// TwinCAT 3 PLC project Machine
// Title: test
// Company: test
// ProjectVersion: 1.1
// ProgramVersion: 3.1.4022.1
// libraries:
//   GWP Library, * (Viessmann)
//   Tc2_Standard, * (Beckhoff Automation GmbH)
//   Tc2_System, * (Beckhoff Automation GmbH)
//   Tc3_Module, * (Beckhoff Automation GmbH)
//   VisuDialogs, * (System)
//   VisuSymbols, * (System)
//   VisuSymbols,3.5.10.0,System
// project tree:
//   / GlobalTextList.TcGTLO, PlcTask.TcTTO, VisualizationManager.TcVMO (not stored), VISU_TASK.TcTTO
//   POUs/ IOs.TcPOU, Main.TcPOU
//   VISUs/ Infoseite.TcVIS, Alarmliste.TcVIS, Fusszeile_50.TcVIS, Test_Login.TcVIS, Testkachel.TcVIS
//   VISUs/Benutzerebene/ Login.TcVIS
//   VISUs/Betriebsarten/Wärmegewinnung/KWP/ KWP_SP_AC_NC_CLK_D.TcVIS, KWP_SP_AC_NC.TcVIS, KWP_SP_AC_NC_GR_4_ohne_RE.TcVIS, KWP_SP_AC_NC_Sollwerte.TcVIS, KWP_SP_AC_NC_PU_Sollwerte.TcVIS
//   VISUs/Betriebsarten/Wärmegewinnung/VD/ VD_Sollwerte_zuruecksetzen.TcVIS, VD.TcVIS, VD_GW_Sollwerte.TcVIS, VD_PU_Sollwerte.TcVIS, VD_VTL_Sollwerte.TcVIS
//   VISUs/Betriebsarten/Wärmesenke/HWP_SP/ HWP_SP.TcVIS, HWP_SP_CLK_D.TcVIS, HWP_SP_GR_4_ohne_RE.TcVIS, HWP_SP_Sollwerte.TcVIS
//   VISUs/Betriebsarten/Wärmesenke/KD/ KD.TcVIS, KD_PU_Sollwerte.TcVIS, KD_Sollwerte_zuruecksetzen.TcVIS, KD_VTL_Sollwerte.TcVIS
//   VISUs/Betriebsarten/Wärmesenke/TWW_SP/ TWW_SP.TcVIS, TWW_SP_CLK_I_Zwangsladung_1.TcVIS, TWW_SP_Sollwerte.TcVIS, TWW_SP_CLK_I_Zwangsladung_2.TcVIS, TWW_SP_PU_Sollwerte.TcVIS
//   VISUs/Betriebsarten/Wärmesenke/Zirkulationspumpe/ Zirkulationspumpe_Sollwerte.TcVIS, Zirkulationspumpe_CLK_W7_Siebentageprogramm.TcVIS
//   VISUs/Betriebsarten/Wärmesenke/Zusatzheizung/ Zusatzheizung_Sollwerte.TcVIS
//   VISUs/Hauptmenu/ Hauptmenu.TcVIS
//   VISUs/Home/ Home.TcVIS
//   VISUs/Maschine/ EG_Innen.TcVIS, EEv.TcVIS, Kreis_3KO_SollwerteAllg.TcVIS, Kreis_3KO.TcVIS
//   VISUs/Sollwertmenu/ Sollwertmenu.TcVIS, Sollwertmenu_Zirk_PU.TcVIS, Sollwertmenu_Waermegewinnung.TcVIS, Sollwertmenu_Waermepumpe.TcVIS, Sollwertmenu_KWP.TcVIS, Sollwertmenu_Waermesenke.TcVIS, Sollwertmenu_KD.TcVIS, Sollwertmenu_HWP.TcVIS, Sollwertmenu_TWW.TcVIS
// real-time tasks:
//   TASK PlcTask: cycle T#10ms, priority 20, ADS port 350
//   TASK VISU_TASK: cycle T#200000us, priority 30, ADS port 351
// I/O:
//   DEVICE Device 1 (EtherCAT), AmsNetId 5.52.29.192.2.1
//     Term 1 (EK1100) [EK1100 EtherCAT Coupler (2A E-Bus)]
//       Term 2 (EL1809) [EL1809 16Ch. Dig. Input 24V, 3ms]
//       Term 3 (EL2809) [EL2809 16Ch. Dig. Output 24V, 0.5A]
//       Term 4 (EL3208) [EL3208 8Ch. Ana. Input PT100 (RTD)]
//       Term 5 (EL3208) [EL3208 8Ch. Ana. Input PT100 (RTD)]
//       Term 6 (EL3058) [EL3058 8Ch. Ana. Input 4-20mA]
//       Term 7 (EL4008) [EL4008 8Ch. Ana. Output 0-10V, 12bit]
//       Term 8 (EL7031) [EL7031 1Ch. Stepper motor output stage (24V, 1.5A)]
//       Term 9 (EL1809) [EL1809 16Ch. Dig. Input 24V, 3ms]
//       Term 10 (EL1809) [EL1809 16Ch. Dig. Input 24V, 3ms]
//       Term 11 (EL2809) [EL2809 16Ch. Dig. Output 24V, 0.5A]
//       Term 12 (EL2809) [EL2809 16Ch. Dig. Output 24V, 0.5A]
//       Term 13 (EL3208) [EL3208 8Ch. Ana. Input PT100 (RTD)]
//       Term 14 (EL3208) [EL3208 8Ch. Ana. Input PT100 (RTD)]
//       Term 15 (EL4008) [EL4008 8Ch. Ana. Output 0-10V, 12bit]
//       Term 16 (EL3208) [EL3208 8Ch. Ana. Input PT100 (RTD)]
//       Term 17 (EL3403-0010) [EL3403-0010 3Ch. Power Measuring, 5A]
//       Term 18 (EL9011) [EL9011 End Terminal]
// variable links:
//   Machine/Machine Instance <-> Device 1 (EtherCAT)/Term 1 (EK1100)/Term 10 (EL1809)
//     PlcTask Inputs/Main.IOs_0.DI_851KF1.ix_DI{1..16} <-> Channel {1..16}/Input  (16 links)
//   Machine/Machine Instance <-> Device 1 (EtherCAT)/Term 1 (EK1100)/Term 11 (EL2809)
//     PlcTask Outputs/Main.IOs_0.DO_851KF2.qx_DO{1..16} <-> Channel {1..16}/Output  (16 links)
//   Machine/Machine Instance <-> Device 1 (EtherCAT)/Term 1 (EK1100)/Term 12 (EL2809)
//     PlcTask Outputs/Main.IOs_0.DO_851KF2_1.qx_DO{1..16} <-> Channel {1..16}/Output  (16 links)
//   Machine/Machine Instance <-> Device 1 (EtherCAT)/Term 1 (EK1100)/Term 13 (EL3208)
//     PlcTask Inputs/Main.IOs_0.AI_851KF3.ii_AI{1..8} <-> RTD Inputs Channel {1..8}/Value  (8 links)
//   Machine/Machine Instance <-> Device 1 (EtherCAT)/Term 1 (EK1100)/Term 14 (EL3208)
//     PlcTask Inputs/Main.IOs_0.AI_851KF4.ii_AI{1..8} <-> RTD Inputs Channel {1..8}/Value  (8 links)
//   Machine/Machine Instance <-> Device 1 (EtherCAT)/Term 1 (EK1100)/Term 15 (EL4008)
//     PlcTask Outputs/Main.IOs_0.AO_851KF4_1.qi_AO{1..8} <-> AO Outputs Channel {1..8}/Analog output  (8 links)
//   Machine/Machine Instance <-> Device 1 (EtherCAT)/Term 1 (EK1100)/Term 16 (EL3208)
//     PlcTask Inputs/Main.IOs_0.AI_851KF6.ii_AI{1..8} <-> RTD Inputs Channel {1..8}/Value  (8 links)
//   Machine/Machine Instance <-> Device 1 (EtherCAT)/Term 1 (EK1100)/Term 17 (EL3403-0010)
//     PlcTask Inputs/Main.IOs_0.EM_851KF6_1.ii_ActivePower_L1 <-> PM Inputs Channel 1/Active power
//     PlcTask Inputs/Main.IOs_0.EM_851KF6_1.ii_ActivePower_L2 <-> PM Inputs Channel 2/Active power
//     PlcTask Inputs/Main.IOs_0.EM_851KF6_1.ii_ActivePower_L3 <-> PM Inputs Channel 3/Active power
//     PlcTask Inputs/Main.IOs_0.EM_851KF6_1.ii_Current_L1 <-> PM Inputs Channel 1/Current
//     PlcTask Inputs/Main.IOs_0.EM_851KF6_1.ii_Current_L2 <-> PM Inputs Channel 2/Current
//     PlcTask Inputs/Main.IOs_0.EM_851KF6_1.ii_Current_L3 <-> PM Inputs Channel 3/Current
//     PlcTask Inputs/Main.IOs_0.EM_851KF6_1.ii_Index_L1 <-> PM Inputs Channel 1/Index
//     PlcTask Inputs/Main.IOs_0.EM_851KF6_1.ii_Index_L2 <-> PM Inputs Channel 2/Index
//     PlcTask Inputs/Main.IOs_0.EM_851KF6_1.ii_Index_L3 <-> PM Inputs Channel 3/Index
//     PlcTask Inputs/Main.IOs_0.EM_851KF6_1.ii_VariantValue_L1 <-> PM Inputs Channel 1/Variant value
//     PlcTask Inputs/Main.IOs_0.EM_851KF6_1.ii_VariantValue_L2 <-> PM Inputs Channel 2/Variant value
//     PlcTask Inputs/Main.IOs_0.EM_851KF6_1.ii_VariantValue_L3 <-> PM Inputs Channel 3/Variant value
//     PlcTask Inputs/Main.IOs_0.EM_851KF6_1.ii_Voltage_L1 <-> PM Inputs Channel 1/Voltage
//     PlcTask Inputs/Main.IOs_0.EM_851KF6_1.ii_Voltage_L2 <-> PM Inputs Channel 2/Voltage
//     PlcTask Inputs/Main.IOs_0.EM_851KF6_1.ii_Voltage_L3 <-> PM Inputs Channel 3/Voltage
//     PlcTask Outputs/Main.IOs_0.EM_851KF6_1.qi_Index_L1 <-> PM Outputs Channel 1/Index
//     PlcTask Outputs/Main.IOs_0.EM_851KF6_1.qi_Index_L2 <-> PM Outputs Channel 2/Index
//     PlcTask Outputs/Main.IOs_0.EM_851KF6_1.qi_Index_L3 <-> PM Outputs Channel 3/Index
//   Machine/Machine Instance <-> Device 1 (EtherCAT)/Term 1 (EK1100)/Term 2 (EL1809)
//     PlcTask Inputs/Main.IOs_0.DI_850KF2.ix_DI{1..16} <-> Channel {1..16}/Input  (16 links)
//   Machine/Machine Instance <-> Device 1 (EtherCAT)/Term 1 (EK1100)/Term 3 (EL2809)
//     PlcTask Outputs/Main.IOs_0.DO_850KF3.qx_DO{1..16} <-> Channel {1..16}/Output  (16 links)
//   Machine/Machine Instance <-> Device 1 (EtherCAT)/Term 1 (EK1100)/Term 4 (EL3208)
//     PlcTask Inputs/Main.IOs_0.AI_850KF4.ii_AI{1..8} <-> RTD Inputs Channel {1..8}/Value  (8 links)
//   Machine/Machine Instance <-> Device 1 (EtherCAT)/Term 1 (EK1100)/Term 5 (EL3208)
//     PlcTask Inputs/Main.IOs_0.AI_850KF4_1.ii_AI{1..8} <-> RTD Inputs Channel {1..8}/Value  (8 links)
//   Machine/Machine Instance <-> Device 1 (EtherCAT)/Term 1 (EK1100)/Term 6 (EL3058)
//     PlcTask Inputs/Main.IOs_0.AI_850KF5.ii_AI{1..8} <-> AI Standard Channel {1..8}/Value  (8 links)
//   Machine/Machine Instance <-> Device 1 (EtherCAT)/Term 1 (EK1100)/Term 7 (EL4008)
//     PlcTask Outputs/Main.IOs_0.AO_850KF6.qi_AO{1..8} <-> AO Outputs Channel {1..8}/Analog output  (8 links)
//   Machine/Machine Instance <-> Device 1 (EtherCAT)/Term 1 (EK1100)/Term 8 (EL7031)
//     PlcTask Inputs/Main.IOs_0.SM_850KF6_1.ii_CounterValue <-> ENC Status/Counter value
//     PlcTask Outputs/Main.IOs_0.SM_850KF6_1.qi_SetCounter <-> ENC Control/Set counter value
//     PlcTask Outputs/Main.IOs_0.SM_850KF6_1.qi_Velo <-> STM Velocity/Velocity
//     PlcTask Outputs/Main.IOs_0.SM_850KF6_1.qx_EN <-> STM Control/Control/Enable
//     PlcTask Outputs/Main.IOs_0.SM_850KF6_1.qx_SetCounter <-> ENC Control/Control/Set counter
//   Machine/Machine Instance <-> Device 1 (EtherCAT)/Term 1 (EK1100)/Term 9 (EL1809)
//     PlcTask Inputs/Main.IOs_0.DI_851KF0.ix_DI{1..16} <-> Channel {1..16}/Input  (16 links)

CONFIGURATION Machine
    RESOURCE PLC ON TwinCAT3
        TASK PlcTask(INTERVAL := T#10ms, PRIORITY := 20);
        TASK VISU_TASK(INTERVAL := T#200000us, PRIORITY := 30);
        PROGRAM Main WITH PlcTask : Main;
        PROGRAM VisuElems_Visu_Prg WITH VISU_TASK : VisuElems.Visu_Prg;
    END_RESOURCE
END_CONFIGURATION

// ---- POUs/Main.TcPOU
PROGRAM Main
VAR
	KWP_SP_AC_NC_0: KWP_SP_AC_NC;
	VD_0: VD;
	KD_0: KD;
	Kreis_3KO_0: Kreis_3KO;
	HWP_SP_0: HWP_SP;
	Zusatzheizung_0: Zusatzheizung;
	Zirk_Pumpe_0: Zirk_Pumpe;
	TWW_SP_0: TWW_SP;
	Init_0: Init;
	IOs_0: IOs;
	AI_to_Druck_0: AI_to_Druck;
	AI_to_Druck_1: AI_to_Druck;
	Logger_0: logger;
	Alarme_1bis10: alarm;
	Alarme_11bis20: alarm;
	Alarme_21bis30: alarm;
	Alarmliste_FB_0: Alarmliste_FB;
END_VAR
VAR PERSISTENT
	dut_Liste:SW_Struct;
END_VAR

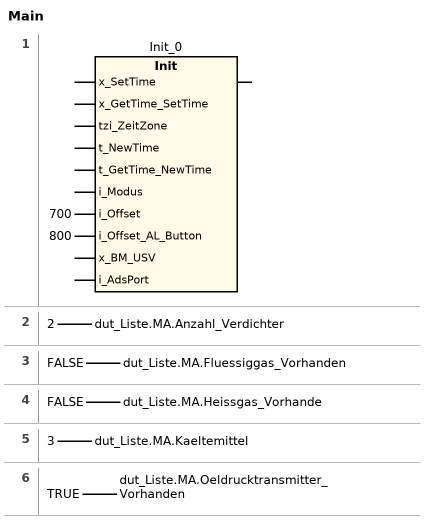
// NETWORK 1
Init_0(i_Offset := 700, i_Offset_AL_Button := 800); // Init

// NETWORK 2
dut_Liste.MA.Anzahl_Verdichter := 2;

// NETWORK 3
dut_Liste.MA.Fluessiggas_Vorhanden := FALSE;

// NETWORK 4
dut_Liste.MA.Heissgas_Vorhande := FALSE;

// NETWORK 5
dut_Liste.MA.Kaeltemittel := 3;

// NETWORK 6
dut_Liste.MA.Oeldrucktransmitter_Vorhanden := TRUE;

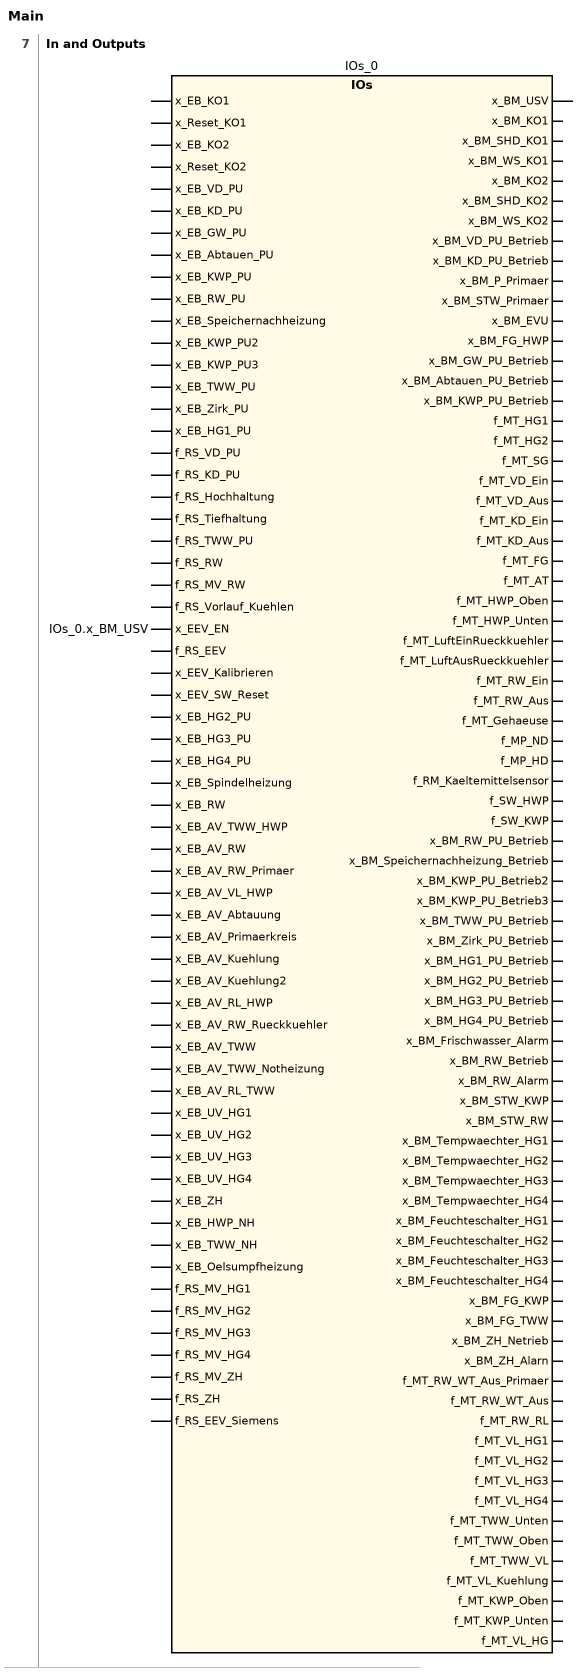
// NETWORK 7: In and Outputs
IOs_0(x_EEV_EN := IOs_0.x_BM_USV); // IOs

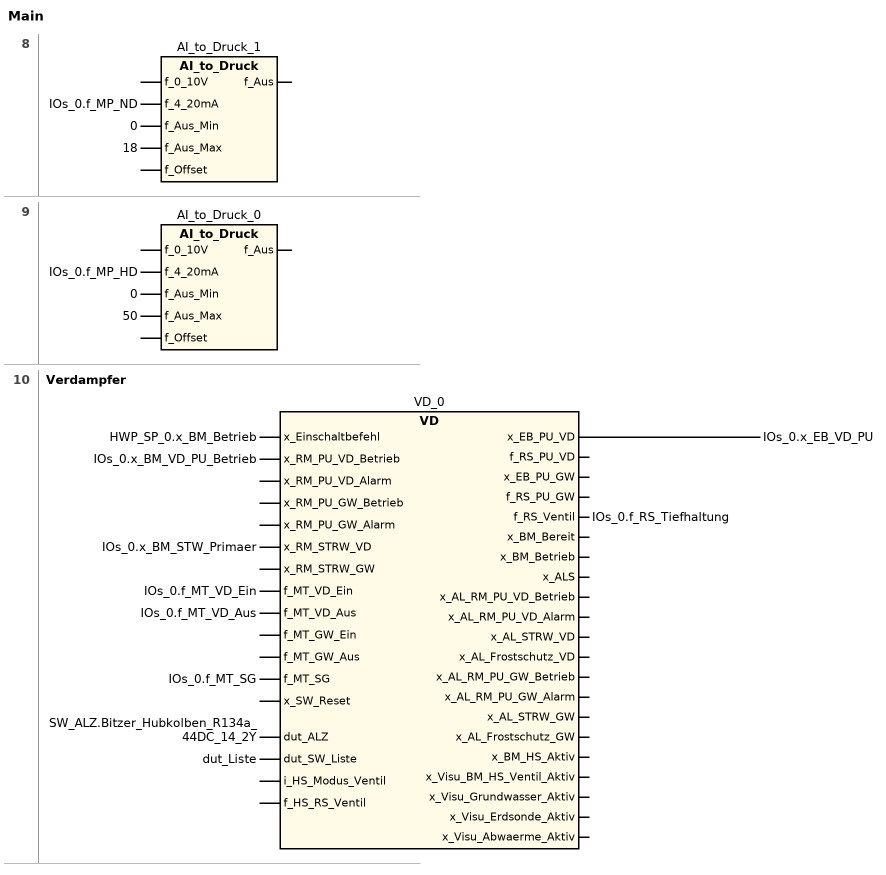
// NETWORK 8
AI_to_Druck_1(f_4_20mA := IOs_0.f_MP_ND, f_Aus_Min := 0, f_Aus_Max := 18); // AI_to_Druck

// NETWORK 9
AI_to_Druck_0(f_4_20mA := IOs_0.f_MP_HD, f_Aus_Min := 0, f_Aus_Max := 50); // AI_to_Druck

// NETWORK 10: Verdampfer
VD_0(
    x_Einschaltbefehl := HWP_SP_0.x_BM_Betrieb,
    x_RM_PU_VD_Betrieb := IOs_0.x_BM_VD_PU_Betrieb,
    x_RM_STRW_VD := IOs_0.x_BM_STW_Primaer,
    f_MT_VD_Ein := IOs_0.f_MT_VD_Ein,
    f_MT_VD_Aus := IOs_0.f_MT_VD_Aus,
    f_MT_SG := IOs_0.f_MT_SG,
    dut_ALZ := SW_ALZ.Bitzer_Hubkolben_R134a_44DC_14_2Y,
    dut_SW_Liste := dut_Liste,
    f_RS_Ventil => IOs_0.f_RS_Tiefhaltung); // VD
IOs_0.x_EB_VD_PU := VD_0.x_EB_PU_VD;

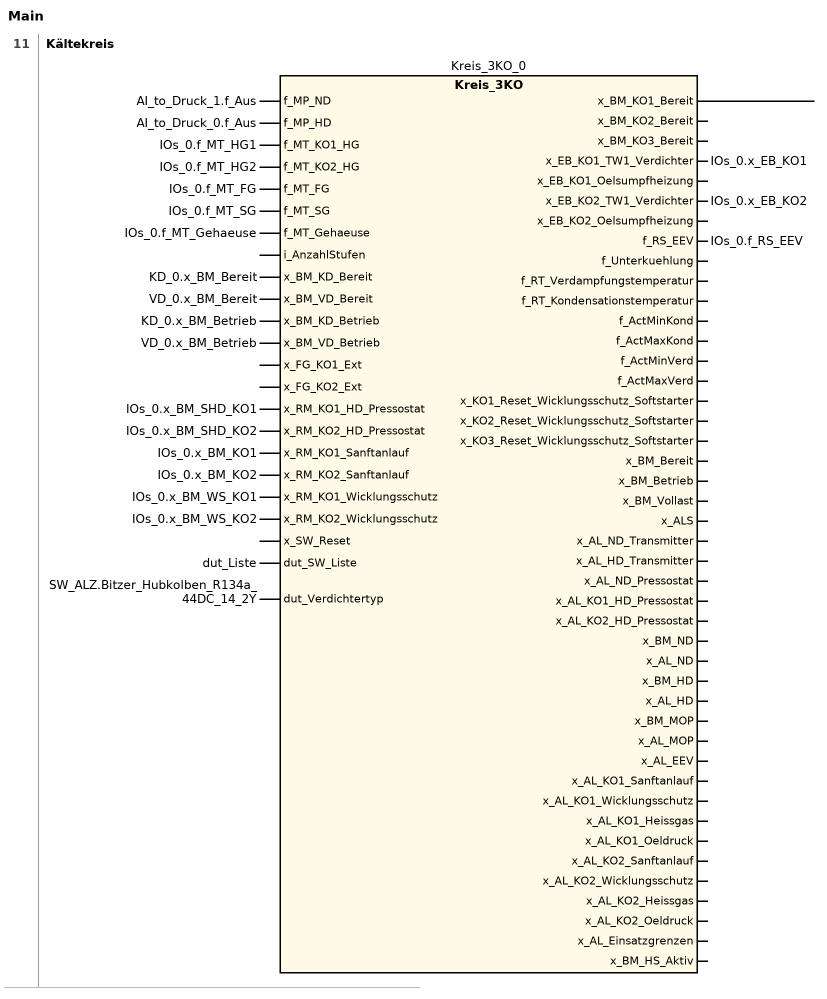
// NETWORK 11: Kältekreis
Kreis_3KO_0(
    f_MP_ND := AI_to_Druck_1.f_Aus,
    f_MP_HD := AI_to_Druck_0.f_Aus,
    f_MT_KO1_HG := IOs_0.f_MT_HG1,
    f_MT_KO2_HG := IOs_0.f_MT_HG2,
    f_MT_FG := IOs_0.f_MT_FG,
    f_MT_SG := IOs_0.f_MT_SG,
    f_MT_Gehaeuse := IOs_0.f_MT_Gehaeuse,
    x_BM_KD_Bereit := KD_0.x_BM_Bereit,
    x_BM_VD_Bereit := VD_0.x_BM_Bereit,
    x_BM_KD_Betrieb := KD_0.x_BM_Betrieb,
    x_BM_VD_Betrieb := VD_0.x_BM_Betrieb,
    x_RM_KO1_HD_Pressostat := IOs_0.x_BM_SHD_KO1,
    x_RM_KO2_HD_Pressostat := IOs_0.x_BM_SHD_KO2,
    x_RM_KO1_Sanftanlauf := IOs_0.x_BM_KO1,
    x_RM_KO2_Sanftanlauf := IOs_0.x_BM_KO2,
    x_RM_KO1_Wicklungsschutz := IOs_0.x_BM_WS_KO1,
    x_RM_KO2_Wicklungsschutz := IOs_0.x_BM_WS_KO2,
    dut_SW_Liste := dut_Liste,
    dut_Verdichtertyp := SW_ALZ.Bitzer_Hubkolben_R134a_44DC_14_2Y,
    x_EB_KO1_TW1_Verdichter => IOs_0.x_EB_KO1,
    x_EB_KO2_TW1_Verdichter => IOs_0.x_EB_KO2,
    f_RS_EEV => IOs_0.f_RS_EEV); // Kreis_3KO

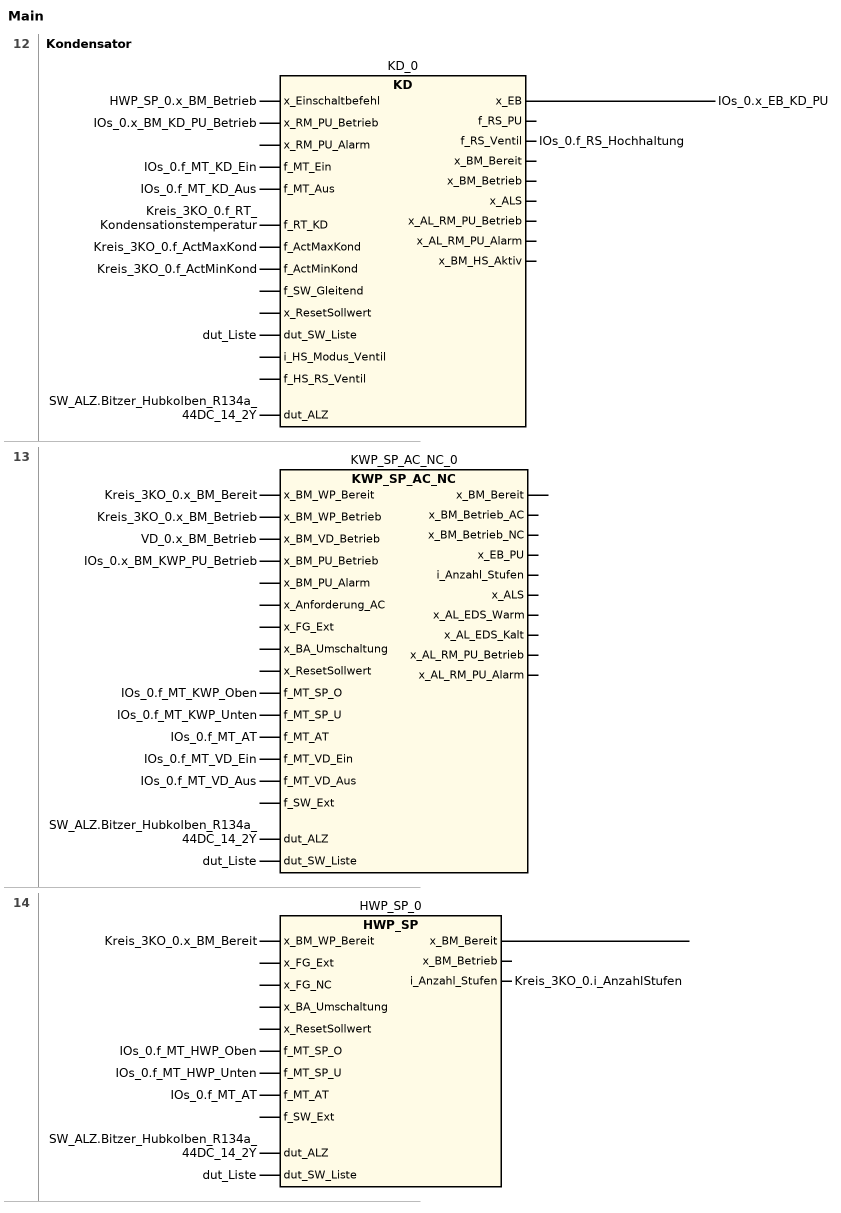
// NETWORK 12: Kondensator
KD_0(
    x_Einschaltbefehl := HWP_SP_0.x_BM_Betrieb,
    x_RM_PU_Betrieb := IOs_0.x_BM_KD_PU_Betrieb,
    f_MT_Ein := IOs_0.f_MT_KD_Ein,
    f_MT_Aus := IOs_0.f_MT_KD_Aus,
    f_RT_KD := Kreis_3KO_0.f_RT_Kondensationstemperatur,
    f_ActMaxKond := Kreis_3KO_0.f_ActMaxKond,
    f_ActMinKond := Kreis_3KO_0.f_ActMinKond,
    dut_SW_Liste := dut_Liste,
    dut_ALZ := SW_ALZ.Bitzer_Hubkolben_R134a_44DC_14_2Y,
    f_RS_Ventil => IOs_0.f_RS_Hochhaltung); // KD
IOs_0.x_EB_KD_PU := KD_0.x_EB;

// NETWORK 13
KWP_SP_AC_NC_0(
    x_BM_WP_Bereit := Kreis_3KO_0.x_BM_Bereit,
    x_BM_WP_Betrieb := Kreis_3KO_0.x_BM_Betrieb,
    x_BM_VD_Betrieb := VD_0.x_BM_Betrieb,
    x_BM_PU_Betrieb := IOs_0.x_BM_KWP_PU_Betrieb,
    f_MT_SP_O := IOs_0.f_MT_KWP_Oben,
    f_MT_SP_U := IOs_0.f_MT_KWP_Unten,
    f_MT_AT := IOs_0.f_MT_AT,
    f_MT_VD_Ein := IOs_0.f_MT_VD_Ein,
    f_MT_VD_Aus := IOs_0.f_MT_VD_Aus,
    dut_ALZ := SW_ALZ.Bitzer_Hubkolben_R134a_44DC_14_2Y,
    dut_SW_Liste := dut_Liste); // KWP_SP_AC_NC

// NETWORK 14
HWP_SP_0(
    x_BM_WP_Bereit := Kreis_3KO_0.x_BM_Bereit,
    f_MT_SP_O := IOs_0.f_MT_HWP_Oben,
    f_MT_SP_U := IOs_0.f_MT_HWP_Unten,
    f_MT_AT := IOs_0.f_MT_AT,
    dut_ALZ := SW_ALZ.Bitzer_Hubkolben_R134a_44DC_14_2Y,
    dut_SW_Liste := dut_Liste,
    i_Anzahl_Stufen => Kreis_3KO_0.i_AnzahlStufen); // HWP_SP

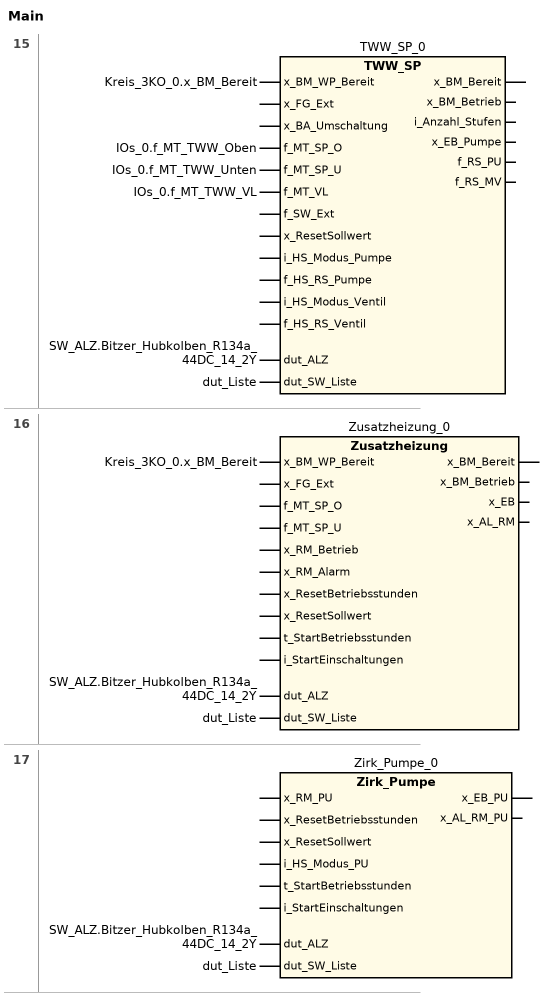
// NETWORK 15
TWW_SP_0(
    x_BM_WP_Bereit := Kreis_3KO_0.x_BM_Bereit,
    f_MT_SP_O := IOs_0.f_MT_TWW_Oben,
    f_MT_SP_U := IOs_0.f_MT_TWW_Unten,
    f_MT_VL := IOs_0.f_MT_TWW_VL,
    dut_ALZ := SW_ALZ.Bitzer_Hubkolben_R134a_44DC_14_2Y,
    dut_SW_Liste := dut_Liste); // TWW_SP

// NETWORK 16
Zusatzheizung_0(
    x_BM_WP_Bereit := Kreis_3KO_0.x_BM_Bereit,
    dut_ALZ := SW_ALZ.Bitzer_Hubkolben_R134a_44DC_14_2Y,
    dut_SW_Liste := dut_Liste); // Zusatzheizung

// NETWORK 17
Zirk_Pumpe_0(dut_ALZ := SW_ALZ.Bitzer_Hubkolben_R134a_44DC_14_2Y, dut_SW_Liste := dut_Liste); // Zirk_Pumpe

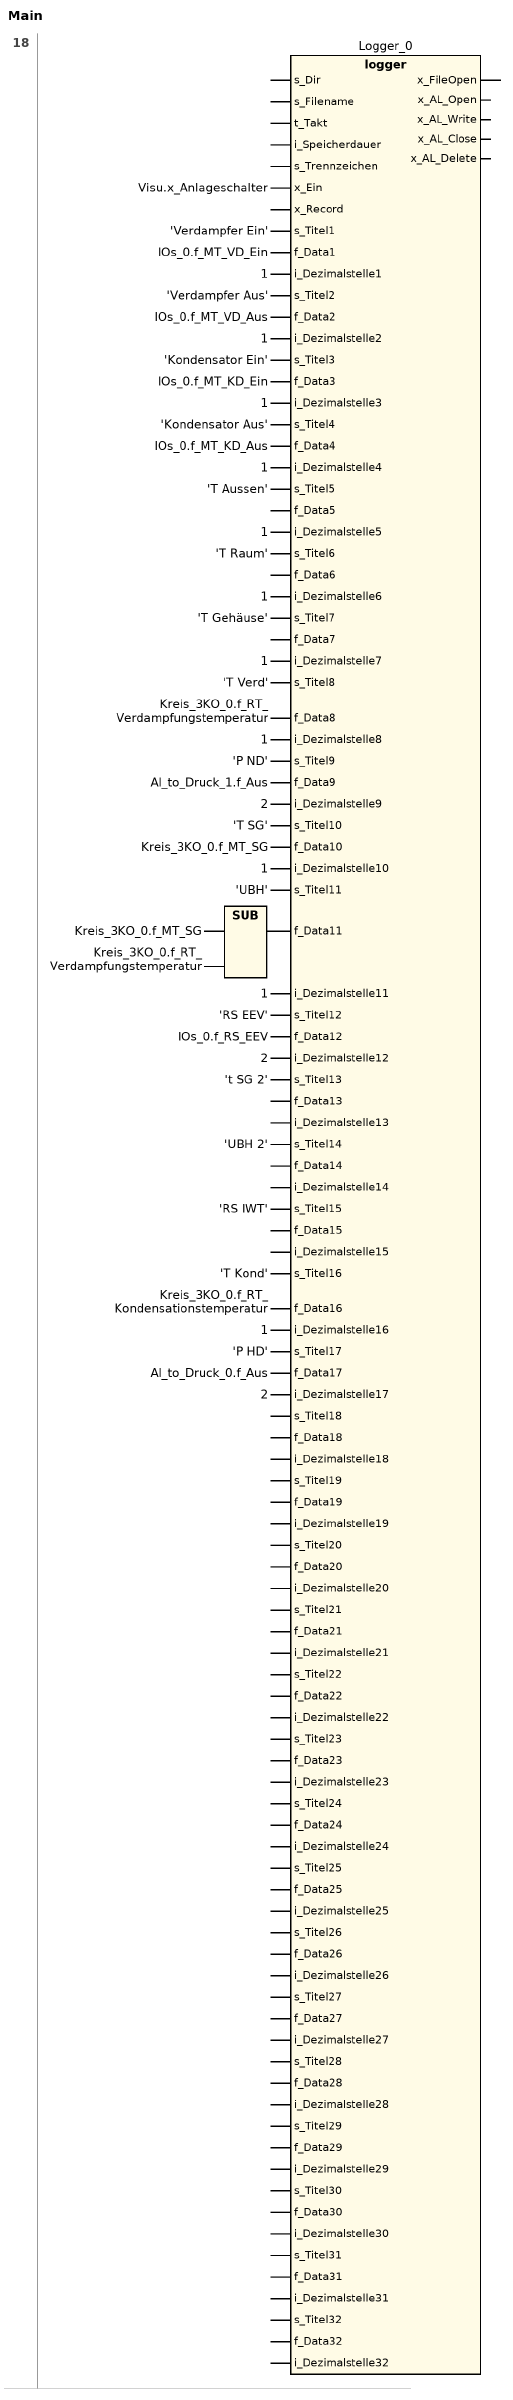
// NETWORK 18
Logger_0(
    x_Ein := Visu.x_Anlageschalter,
    s_Titel1 := 'Verdampfer Ein',
    f_Data1 := IOs_0.f_MT_VD_Ein,
    i_Dezimalstelle1 := 1,
    s_Titel2 := 'Verdampfer Aus',
    f_Data2 := IOs_0.f_MT_VD_Aus,
    i_Dezimalstelle2 := 1,
    s_Titel3 := 'Kondensator Ein',
    f_Data3 := IOs_0.f_MT_KD_Ein,
    i_Dezimalstelle3 := 1,
    s_Titel4 := 'Kondensator Aus',
    f_Data4 := IOs_0.f_MT_KD_Aus,
    i_Dezimalstelle4 := 1,
    s_Titel5 := 'T Aussen',
    i_Dezimalstelle5 := 1,
    s_Titel6 := 'T Raum',
    i_Dezimalstelle6 := 1,
    s_Titel7 := 'T Gehäuse',
    i_Dezimalstelle7 := 1,
    s_Titel8 := 'T Verd',
    f_Data8 := Kreis_3KO_0.f_RT_Verdampfungstemperatur,
    i_Dezimalstelle8 := 1,
    s_Titel9 := 'P ND',
    f_Data9 := AI_to_Druck_1.f_Aus,
    i_Dezimalstelle9 := 2,
    s_Titel10 := 'T SG',
    f_Data10 := Kreis_3KO_0.f_MT_SG,
    i_Dezimalstelle10 := 1,
    s_Titel11 := 'UBH',
    f_Data11 := Kreis_3KO_0.f_MT_SG - Kreis_3KO_0.f_RT_Verdampfungstemperatur,
    i_Dezimalstelle11 := 1,
    s_Titel12 := 'RS EEV',
    f_Data12 := IOs_0.f_RS_EEV,
    i_Dezimalstelle12 := 2,
    s_Titel13 := 't SG 2',
    s_Titel14 := 'UBH 2',
    s_Titel15 := 'RS IWT',
    s_Titel16 := 'T Kond',
    f_Data16 := Kreis_3KO_0.f_RT_Kondensationstemperatur,
    i_Dezimalstelle16 := 1,
    s_Titel17 := 'P HD',
    f_Data17 := AI_to_Druck_0.f_Aus,
    i_Dezimalstelle17 := 2); // logger

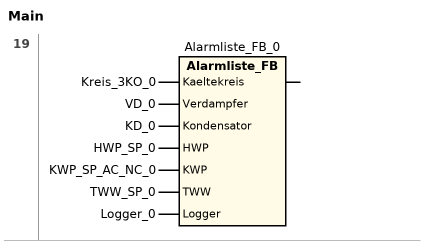
// NETWORK 19
Alarmliste_FB_0(
    Kaeltekreis := Kreis_3KO_0,
    Verdampfer := VD_0,
    Kondensator := KD_0,
    HWP := HWP_SP_0,
    KWP := KWP_SP_AC_NC_0,
    TWW := TWW_SP_0,
    Logger := Logger_0); // Alarmliste_FB

END_PROGRAM

// ---- POUs/IOs.TcPOU
FUNCTION_BLOCK IOs
VAR_INPUT
	//850KF3
	x_EB_KO1: BOOL;
	x_Reset_KO1: BOOL;
	x_EB_KO2: BOOL;
	x_Reset_KO2: BOOL;
	x_EB_VD_PU: BOOL;
	x_EB_KD_PU: BOOL;
	x_EB_GW_PU: BOOL;
	x_EB_Abtauen_PU: BOOL;
	x_EB_KWP_PU: BOOL;
	x_EB_RW_PU: BOOL;
	x_EB_Speichernachheizung: BOOL;
	x_EB_KWP_PU2: BOOL;
	x_EB_KWP_PU3: BOOL;
	x_EB_TWW_PU: BOOL;
	x_EB_Zirk_PU: BOOL;
	x_EB_HG1_PU: BOOL;
	//850KF6
	f_RS_VD_PU: REAL;
	f_RS_KD_PU: REAL;
	f_RS_Hochhaltung: REAL;
	f_RS_Tiefhaltung: REAL;
	f_RS_TWW_PU: REAL;
	f_RS_RW: REAL;
	f_RS_MV_RW: REAL;
	f_RS_Vorlauf_Kuehlen: REAL;
	//850KF6.1
	x_EEV_EN: BOOL;
	f_RS_EEV: REAL;
	x_EEV_Kalibrieren: BOOL;
	x_EEV_SW_Reset: BOOL;
	//851KF2
	x_EB_HG2_PU: BOOL;
	x_EB_HG3_PU: BOOL;
	x_EB_HG4_PU: BOOL;
	x_EB_Spindelheizung: BOOL;
	x_EB_RW: BOOL;
	x_EB_AV_TWW_HWP: BOOL;
	x_EB_AV_RW: BOOL;
	x_EB_AV_RW_Primaer: BOOL;
	x_EB_AV_VL_HWP: BOOL;
	x_EB_AV_Abtauung: BOOL;
	x_EB_AV_Primaerkreis: BOOL;
	x_EB_AV_Kuehlung: BOOL;
	x_EB_AV_Kuehlung2: BOOL;
	x_EB_AV_RL_HWP: BOOL;
	x_EB_AV_RW_Rueckkuehler: BOOL;
	x_EB_AV_TWW: BOOL;
	//851KF2.1
	x_EB_AV_TWW_Notheizung: BOOL;
	x_EB_AV_RL_TWW: BOOL;
	x_EB_UV_HG1: BOOL;
	x_EB_UV_HG2: BOOL;
	x_EB_UV_HG3: BOOL;
	x_EB_UV_HG4: BOOL;
	x_EB_ZH: BOOL;
	x_EB_HWP_NH: BOOL;
	x_EB_TWW_NH: BOOL;
	x_EB_Oelsumpfheizung: BOOL;
	//851KF4.1
	f_RS_MV_HG1: REAL;
	f_RS_MV_HG2: REAL;
	f_RS_MV_HG3: REAL;
	f_RS_MV_HG4: REAL;
	f_RS_MV_ZH: REAL;
	f_RS_ZH: REAL;
	f_RS_EEV_Siemens: REAL;
END_VAR
VAR_OUTPUT
	//850KF2
	x_BM_USV: BOOL;
	x_BM_KO1: BOOL;
	x_BM_SHD_KO1: BOOL;
	x_BM_WS_KO1: BOOL;
	x_BM_KO2: BOOL;
	x_BM_SHD_KO2: BOOL;
	x_BM_WS_KO2: BOOL;
	x_BM_VD_PU_Betrieb: BOOL;
	x_BM_KD_PU_Betrieb: BOOL;
	x_BM_P_Primaer: BOOL;
	x_BM_STW_Primaer: BOOL;
	x_BM_EVU: BOOL;
	x_BM_FG_HWP: BOOL;
	x_BM_GW_PU_Betrieb: BOOL;
	x_BM_Abtauen_PU_Betrieb: BOOL;
	x_BM_KWP_PU_Betrieb: BOOL;
	//850KF4
	f_MT_HG1: REAL;
	f_MT_HG2: REAL;
	f_MT_SG: REAL;
	f_MT_VD_Ein: REAL;
	f_MT_VD_Aus: REAL;
	f_MT_KD_Ein: REAL;
	f_MT_KD_Aus: REAL;
	f_MT_FG: REAL;
	//850KF4.1
	f_MT_AT: REAL;
	f_MT_HWP_Oben: REAL;
	f_MT_HWP_Unten: REAL;
	f_MT_LuftEinRueckkuehler: REAL;
	f_MT_LuftAusRueckkuehler: REAL;
	f_MT_RW_Ein: REAL;
	f_MT_RW_Aus: REAL;
	f_MT_Gehaeuse: REAL;
	//850KF5
	f_MP_ND: REAL;
	f_MP_HD: REAL;
	f_RM_Kaeltemittelsensor: REAL;
	f_SW_HWP: REAL;
	f_SW_KWP: REAL;
	//851KF0
	x_BM_RW_PU_Betrieb: BOOL;
	x_BM_Speichernachheizung_Betrieb: BOOL;
	x_BM_KWP_PU_Betrieb2: BOOL;
	x_BM_KWP_PU_Betrieb3: BOOL;
	x_BM_TWW_PU_Betrieb: BOOL;
	x_BM_Zirk_PU_Betrieb: BOOL;
	x_BM_HG1_PU_Betrieb: BOOL;
	x_BM_HG2_PU_Betrieb: BOOL;
	x_BM_HG3_PU_Betrieb: BOOL;
	x_BM_HG4_PU_Betrieb: BOOL;
	x_BM_Frischwasser_Alarm: BOOL;
	x_BM_RW_Betrieb: BOOL;
	x_BM_RW_Alarm: BOOL;
	x_BM_STW_KWP: BOOL;
	x_BM_STW_RW: BOOL;
	x_BM_Tempwaechter_HG1: BOOL;
	//851KF1
	x_BM_Tempwaechter_HG2: BOOL;
	x_BM_Tempwaechter_HG3: BOOL;
	x_BM_Tempwaechter_HG4: BOOL;
	x_BM_Feuchteschalter_HG1: BOOL;
	x_BM_Feuchteschalter_HG2: BOOL;
	x_BM_Feuchteschalter_HG3: BOOL;
	x_BM_Feuchteschalter_HG4: BOOL;
	x_BM_FG_KWP: BOOL;
	x_BM_FG_TWW: BOOL;
	x_BM_ZH_Netrieb: BOOL;
	x_BM_ZH_Alarn: BOOL;
	//851KF3
	f_MT_RW_WT_Aus_Primaer: REAL;
	f_MT_RW_WT_Aus: REAL;
	f_MT_RW_RL: REAL;
	f_MT_VL_HG1: REAL;
	f_MT_VL_HG2: REAL;
	f_MT_VL_HG3: REAL;
	f_MT_VL_HG4: REAL;
	f_MT_TWW_Unten: REAL;
	//851KF4
	f_MT_TWW_Oben: REAL;
	f_MT_TWW_VL: REAL;
	f_MT_VL_Kuehlung: REAL;
	
	f_MT_KWP_Oben: REAL;
	f_MT_KWP_Unten: REAL;
	f_MT_VL_HG: REAL;
	//851KF6
	
	//851KF6.1
END_VAR
VAR
	DI_850KF2: DI_16;
	DO_850KF3: DO_16;
	AI_850KF4: AI_8_Temp;
	AI_850KF4_1: AI_8_Temp;
	AI_850KF5: AI_8_4_20mA;
	AO_850KF6: AO_8;
	SM_850KF6_1: EEV_Schrittmotor;
	DI_851KF0: DI_16;
	DI_851KF1: DI_16;
	DO_851KF2: DO_16;
	DO_851KF2_1: DO_16;
	AI_851KF3: AI_8_Temp;
	AI_851KF4: AI_8_Temp;
	AO_851KF4_1: AO_8;
	AI_851KF6: AI_8_Temp;
	EM_851KF6_1: Elektromessung;
END_VAR

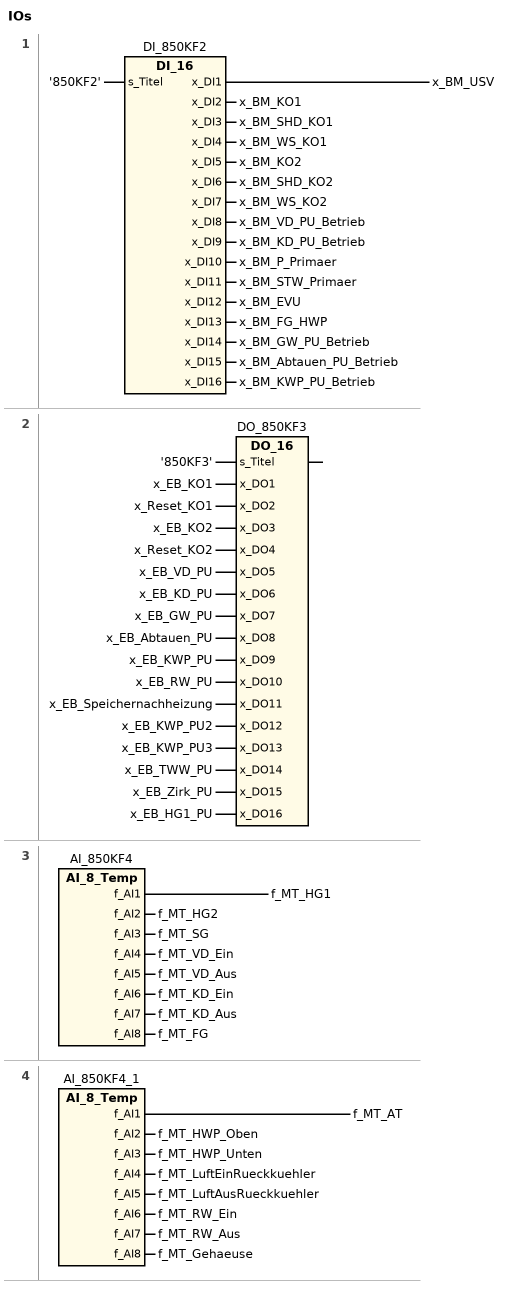
// NETWORK 1
DI_850KF2(
    s_Titel := '850KF2',
    x_DI2 => x_BM_KO1,
    x_DI3 => x_BM_SHD_KO1,
    x_DI4 => x_BM_WS_KO1,
    x_DI5 => x_BM_KO2,
    x_DI6 => x_BM_SHD_KO2,
    x_DI7 => x_BM_WS_KO2,
    x_DI8 => x_BM_VD_PU_Betrieb,
    x_DI9 => x_BM_KD_PU_Betrieb,
    x_DI10 => x_BM_P_Primaer,
    x_DI11 => x_BM_STW_Primaer,
    x_DI12 => x_BM_EVU,
    x_DI13 => x_BM_FG_HWP,
    x_DI14 => x_BM_GW_PU_Betrieb,
    x_DI15 => x_BM_Abtauen_PU_Betrieb,
    x_DI16 => x_BM_KWP_PU_Betrieb); // DI_16
x_BM_USV := DI_850KF2.x_DI1;

// NETWORK 2
DO_850KF3(
    s_Titel := '850KF3',
    x_DO1 := x_EB_KO1,
    x_DO2 := x_Reset_KO1,
    x_DO3 := x_EB_KO2,
    x_DO4 := x_Reset_KO2,
    x_DO5 := x_EB_VD_PU,
    x_DO6 := x_EB_KD_PU,
    x_DO7 := x_EB_GW_PU,
    x_DO8 := x_EB_Abtauen_PU,
    x_DO9 := x_EB_KWP_PU,
    x_DO10 := x_EB_RW_PU,
    x_DO11 := x_EB_Speichernachheizung,
    x_DO12 := x_EB_KWP_PU2,
    x_DO13 := x_EB_KWP_PU3,
    x_DO14 := x_EB_TWW_PU,
    x_DO15 := x_EB_Zirk_PU,
    x_DO16 := x_EB_HG1_PU); // DO_16

// NETWORK 3
AI_850KF4(
    f_AI2 => f_MT_HG2,
    f_AI3 => f_MT_SG,
    f_AI4 => f_MT_VD_Ein,
    f_AI5 => f_MT_VD_Aus,
    f_AI6 => f_MT_KD_Ein,
    f_AI7 => f_MT_KD_Aus,
    f_AI8 => f_MT_FG); // AI_8_Temp
f_MT_HG1 := AI_850KF4.f_AI1;

// NETWORK 4
AI_850KF4_1(
    f_AI2 => f_MT_HWP_Oben,
    f_AI3 => f_MT_HWP_Unten,
    f_AI4 => f_MT_LuftEinRueckkuehler,
    f_AI5 => f_MT_LuftAusRueckkuehler,
    f_AI6 => f_MT_RW_Ein,
    f_AI7 => f_MT_RW_Aus,
    f_AI8 => f_MT_Gehaeuse); // AI_8_Temp
f_MT_AT := AI_850KF4_1.f_AI1;

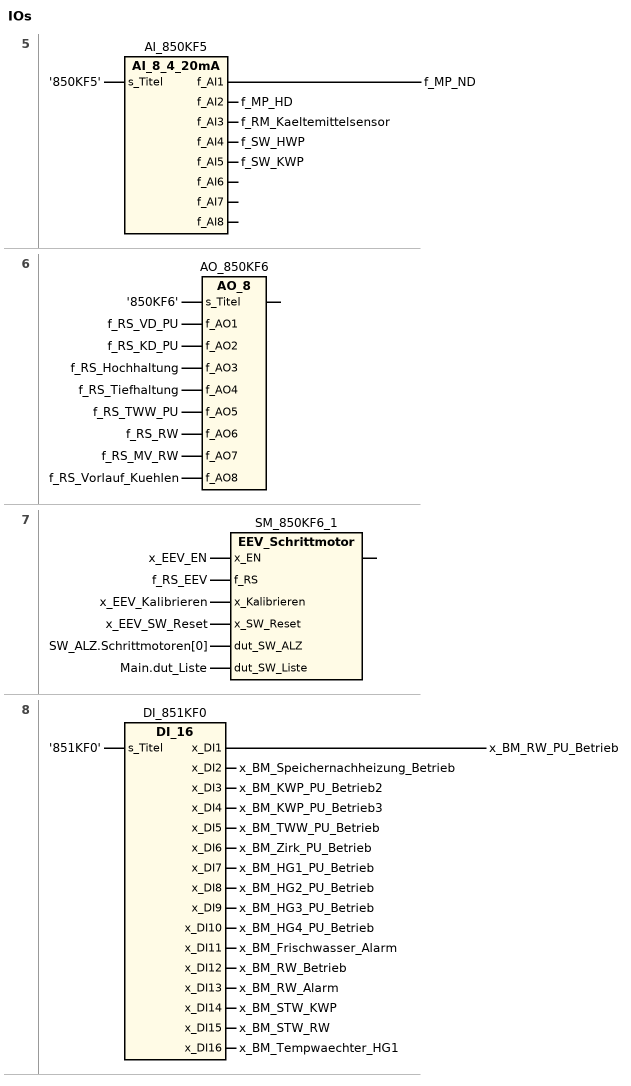
// NETWORK 5
AI_850KF5(
    s_Titel := '850KF5',
    f_AI2 => f_MP_HD,
    f_AI3 => f_RM_Kaeltemittelsensor,
    f_AI4 => f_SW_HWP,
    f_AI5 => f_SW_KWP); // AI_8_4_20mA
f_MP_ND := AI_850KF5.f_AI1;

// NETWORK 6
AO_850KF6(
    s_Titel := '850KF6',
    f_AO1 := f_RS_VD_PU,
    f_AO2 := f_RS_KD_PU,
    f_AO3 := f_RS_Hochhaltung,
    f_AO4 := f_RS_Tiefhaltung,
    f_AO5 := f_RS_TWW_PU,
    f_AO6 := f_RS_RW,
    f_AO7 := f_RS_MV_RW,
    f_AO8 := f_RS_Vorlauf_Kuehlen); // AO_8

// NETWORK 7
SM_850KF6_1(
    x_EN := x_EEV_EN,
    f_RS := f_RS_EEV,
    x_Kalibrieren := x_EEV_Kalibrieren,
    x_SW_Reset := x_EEV_SW_Reset,
    dut_SW_ALZ := SW_ALZ.Schrittmotoren[0],
    dut_SW_Liste := Main.dut_Liste); // EEV_Schrittmotor

// NETWORK 8
DI_851KF0(
    s_Titel := '851KF0',
    x_DI2 => x_BM_Speichernachheizung_Betrieb,
    x_DI3 => x_BM_KWP_PU_Betrieb2,
    x_DI4 => x_BM_KWP_PU_Betrieb3,
    x_DI5 => x_BM_TWW_PU_Betrieb,
    x_DI6 => x_BM_Zirk_PU_Betrieb,
    x_DI7 => x_BM_HG1_PU_Betrieb,
    x_DI8 => x_BM_HG2_PU_Betrieb,
    x_DI9 => x_BM_HG3_PU_Betrieb,
    x_DI10 => x_BM_HG4_PU_Betrieb,
    x_DI11 => x_BM_Frischwasser_Alarm,
    x_DI12 => x_BM_RW_Betrieb,
    x_DI13 => x_BM_RW_Alarm,
    x_DI14 => x_BM_STW_KWP,
    x_DI15 => x_BM_STW_RW,
    x_DI16 => x_BM_Tempwaechter_HG1); // DI_16
x_BM_RW_PU_Betrieb := DI_851KF0.x_DI1;

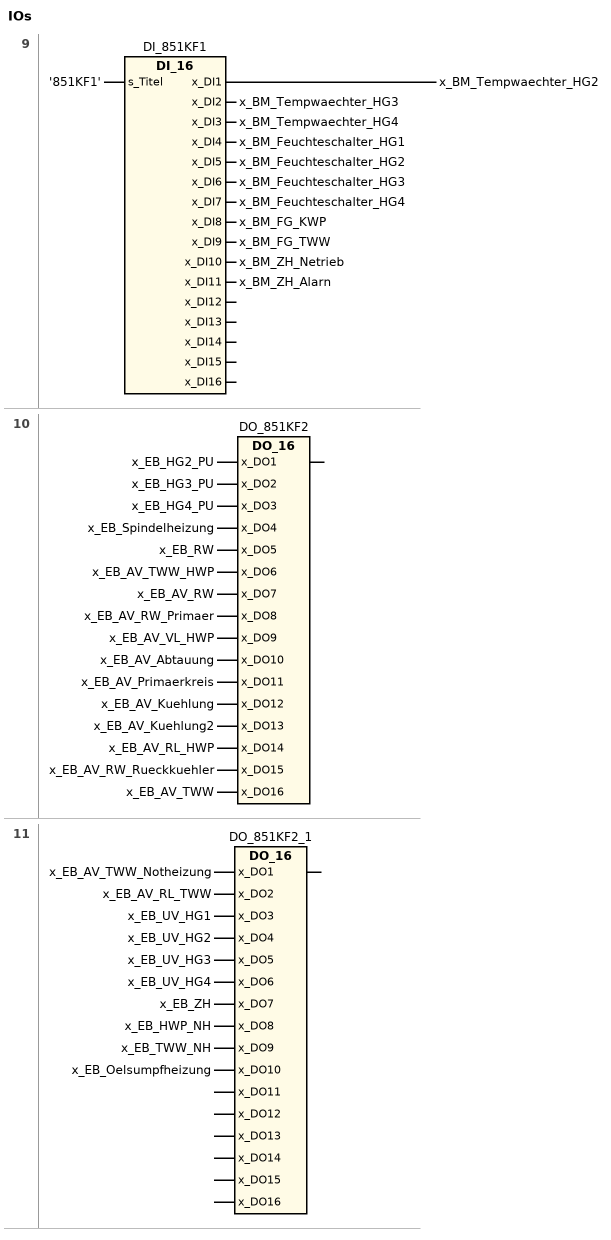
// NETWORK 9
DI_851KF1(
    s_Titel := '851KF1',
    x_DI2 => x_BM_Tempwaechter_HG3,
    x_DI3 => x_BM_Tempwaechter_HG4,
    x_DI4 => x_BM_Feuchteschalter_HG1,
    x_DI5 => x_BM_Feuchteschalter_HG2,
    x_DI6 => x_BM_Feuchteschalter_HG3,
    x_DI7 => x_BM_Feuchteschalter_HG4,
    x_DI8 => x_BM_FG_KWP,
    x_DI9 => x_BM_FG_TWW,
    x_DI10 => x_BM_ZH_Netrieb,
    x_DI11 => x_BM_ZH_Alarn); // DI_16
x_BM_Tempwaechter_HG2 := DI_851KF1.x_DI1;

// NETWORK 10
DO_851KF2(
    x_DO1 := x_EB_HG2_PU,
    x_DO2 := x_EB_HG3_PU,
    x_DO3 := x_EB_HG4_PU,
    x_DO4 := x_EB_Spindelheizung,
    x_DO5 := x_EB_RW,
    x_DO6 := x_EB_AV_TWW_HWP,
    x_DO7 := x_EB_AV_RW,
    x_DO8 := x_EB_AV_RW_Primaer,
    x_DO9 := x_EB_AV_VL_HWP,
    x_DO10 := x_EB_AV_Abtauung,
    x_DO11 := x_EB_AV_Primaerkreis,
    x_DO12 := x_EB_AV_Kuehlung,
    x_DO13 := x_EB_AV_Kuehlung2,
    x_DO14 := x_EB_AV_RL_HWP,
    x_DO15 := x_EB_AV_RW_Rueckkuehler,
    x_DO16 := x_EB_AV_TWW); // DO_16

// NETWORK 11
DO_851KF2_1(
    x_DO1 := x_EB_AV_TWW_Notheizung,
    x_DO2 := x_EB_AV_RL_TWW,
    x_DO3 := x_EB_UV_HG1,
    x_DO4 := x_EB_UV_HG2,
    x_DO5 := x_EB_UV_HG3,
    x_DO6 := x_EB_UV_HG4,
    x_DO7 := x_EB_ZH,
    x_DO8 := x_EB_HWP_NH,
    x_DO9 := x_EB_TWW_NH,
    x_DO10 := x_EB_Oelsumpfheizung); // DO_16

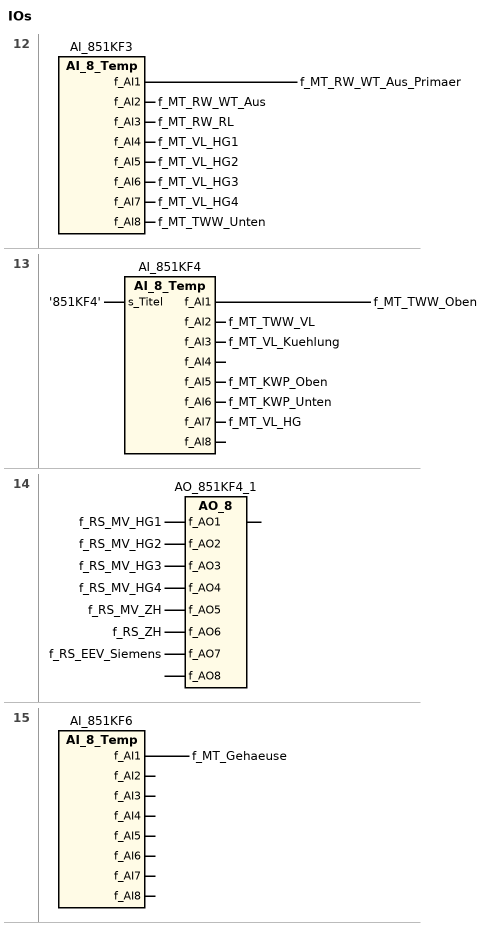
// NETWORK 12
AI_851KF3(
    f_AI2 => f_MT_RW_WT_Aus,
    f_AI3 => f_MT_RW_RL,
    f_AI4 => f_MT_VL_HG1,
    f_AI5 => f_MT_VL_HG2,
    f_AI6 => f_MT_VL_HG3,
    f_AI7 => f_MT_VL_HG4,
    f_AI8 => f_MT_TWW_Unten); // AI_8_Temp
f_MT_RW_WT_Aus_Primaer := AI_851KF3.f_AI1;

// NETWORK 13
AI_851KF4(
    s_Titel := '851KF4',
    f_AI2 => f_MT_TWW_VL,
    f_AI3 => f_MT_VL_Kuehlung,
    f_AI5 => f_MT_KWP_Oben,
    f_AI6 => f_MT_KWP_Unten,
    f_AI7 => f_MT_VL_HG); // AI_8_Temp
f_MT_TWW_Oben := AI_851KF4.f_AI1;

// NETWORK 14
AO_851KF4_1(
    f_AO1 := f_RS_MV_HG1,
    f_AO2 := f_RS_MV_HG2,
    f_AO3 := f_RS_MV_HG3,
    f_AO4 := f_RS_MV_HG4,
    f_AO5 := f_RS_MV_ZH,
    f_AO6 := f_RS_ZH,
    f_AO7 := f_RS_EEV_Siemens); // AO_8

// NETWORK 15
AI_851KF6(); // AI_8_Temp
f_MT_Gehaeuse := AI_851KF6.f_AI1;

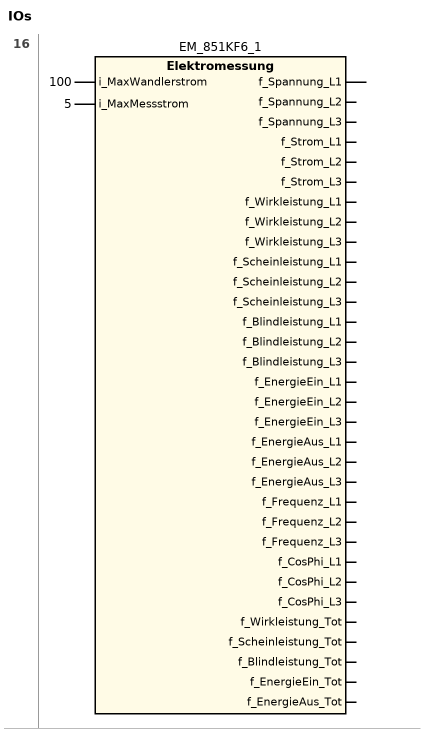
// NETWORK 16
EM_851KF6_1(i_MaxWandlerstrom := 100, i_MaxMessstrom := 5); // Elektromessung

END_FUNCTION_BLOCK

// ---- GlobalTextList.TcGTLO
TEXTLIST GlobalTextList
  978 = '%.1f'
  90 = '%.1f  °C '
  798 = '%.1f K'
  979 = '%.2f'
  607 = '%d.%m.%y'
  68 = '%dd.MM.yy'
  977 = '%i'
  526 = '%i '
  89 = '%s'
  652 = '%t%d.%m.%y'
  527 = ':'
  700 = 'Admin'
  2 = 'ku'
  51 = 'Ku'
  219 = 'Kunde'
  998 = 'Login'
  341 = 'Logiut'
  610 = 'Löschen'
  0 = 'None'
  398 = 'Operator'
  519 = 'Quittieren'
  372 = 'Service'
  766 = 's_Titel'
  91 = 'Techniker'
  1 = 'vi'
  497 = 'Vi'
END_TEXTLIST

// ---- VISUs/Infoseite.TcVIS
VISUALIZATION Infoseite  // 800x480
END_VISUALIZATION

// ---- VISUs/Benutzerebene/Login.TcVIS
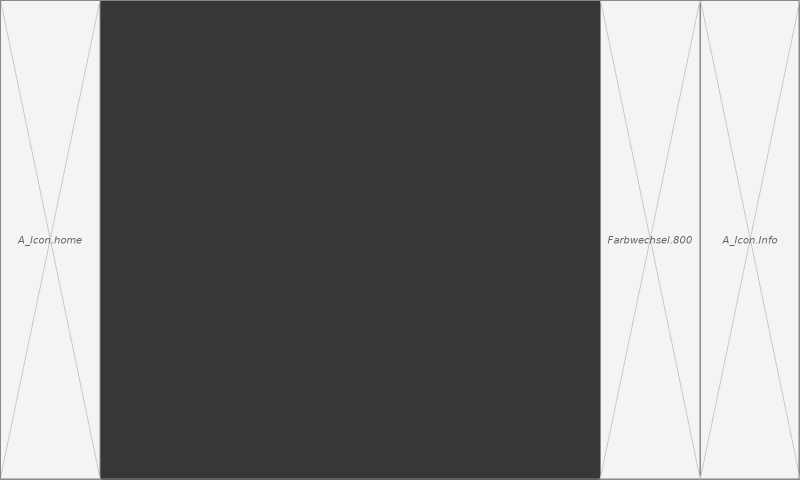
VISUALIZATION Login  // 800x480
    Frame (0,0 800x480)
        shows GWP_Library.Login()
    Frame (0,0 800x480)
        shows Fusszeile_50()
END_VISUALIZATION

// ---- VISUs/Betriebsarten/Wärmegewinnung/KWP/KWP_SP_AC_NC_CLK_D.TcVIS
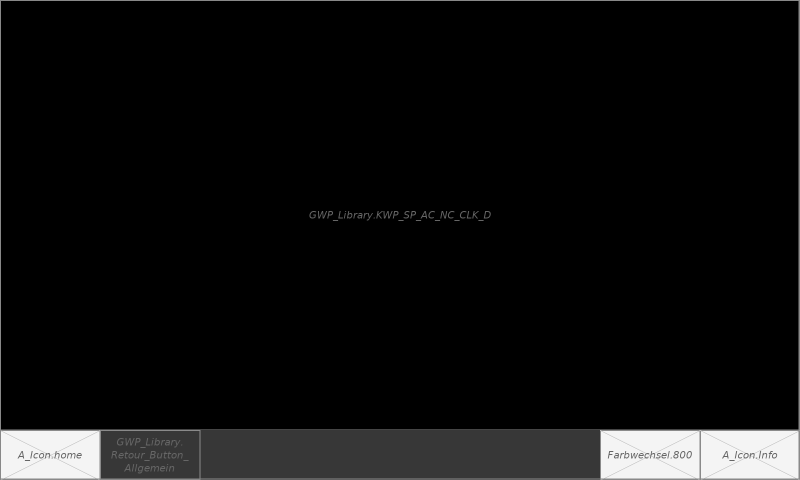
VISUALIZATION KWP_SP_AC_NC_CLK_D  // 800x480
    Frame (0,0 800x430)
        shows GWP_Library.KWP_SP_AC_NC_CLK_D(FB_CLK_D := Main.KWP_SP_AC_NC_0.GR_4_ohne_RE_0.TagNacht)
    Frame (0,430 800x50)
        shows Fusszeile_50()
    Frame (100,430 100x50)
        shows GWP_Library.Retour_Button_Allgemein()
END_VISUALIZATION

// ---- VISUs/Betriebsarten/Wärmegewinnung/KWP/KWP_SP_AC_NC.TcVIS
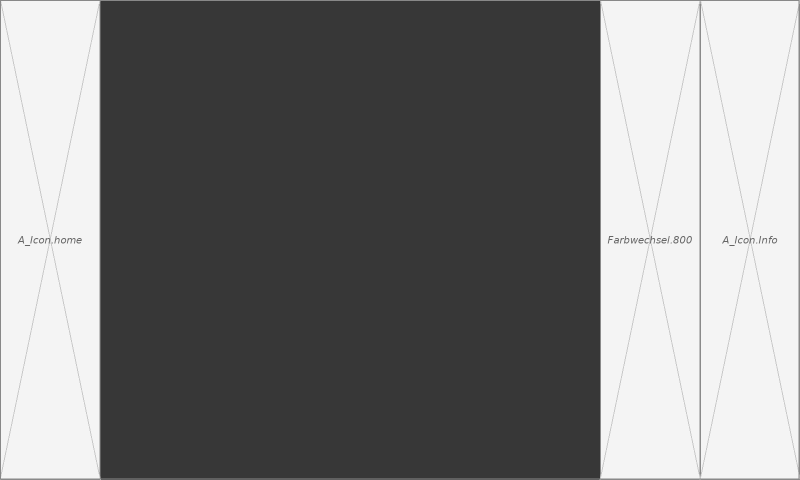
VISUALIZATION KWP_SP_AC_NC  // 800x480
    Frame (0,0 800x430)
        shows GWP_Library.KWP_SP_AC_NC(FB_KWP_SP_AC_NC := Main.KWP_SP_AC_NC_0, FB_Kreis_3KO := Main.Kreis_3KO_0, FB_VD := Main.VD_0)
    Frame (0,0 800x480)
        shows Fusszeile_50()
END_VISUALIZATION

// ---- VISUs/Betriebsarten/Wärmegewinnung/KWP/KWP_SP_AC_NC_GR_4_ohne_RE.TcVIS
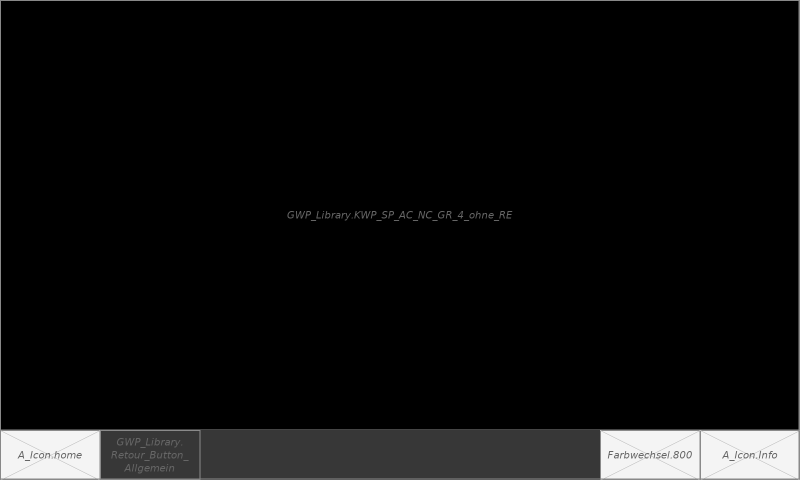
VISUALIZATION KWP_SP_AC_NC_GR_4_ohne_RE  // 800x480
    Frame (0,0 800x430)
        shows GWP_Library.KWP_SP_AC_NC_GR_4_ohne_RE(FB_GR_4_ohne_RE := Main.KWP_SP_AC_NC_0.GR_4_ohne_RE_0)
    Frame (0,430 800x50)
        shows Fusszeile_50()
    Frame (100,430 100x50)
        shows GWP_Library.Retour_Button_Allgemein()
END_VISUALIZATION

// ---- VISUs/Betriebsarten/Wärmegewinnung/KWP/KWP_SP_AC_NC_Sollwerte.TcVIS
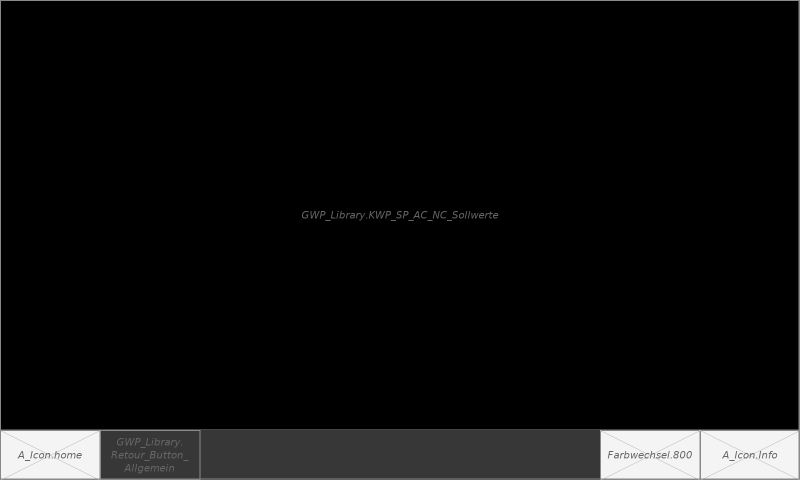
VISUALIZATION KWP_SP_AC_NC_Sollwerte  // 800x480
    Frame (0,0 800x430)
        shows GWP_Library.KWP_SP_AC_NC_Sollwerte(FB_KWP_SP_AC_NC := Main.KWP_SP_AC_NC_0, FB_Kreis_3KO := Main.Kreis_3KO_0, FB_VD := Main.VD_0)
    Frame (0,430 800x50)
        shows Fusszeile_50()
    Frame (100,430 100x50)
        shows GWP_Library.Retour_Button_Allgemein()
END_VISUALIZATION

// ---- VISUs/Betriebsarten/Wärmegewinnung/KWP/KWP_SP_AC_NC_PU_Sollwerte.TcVIS
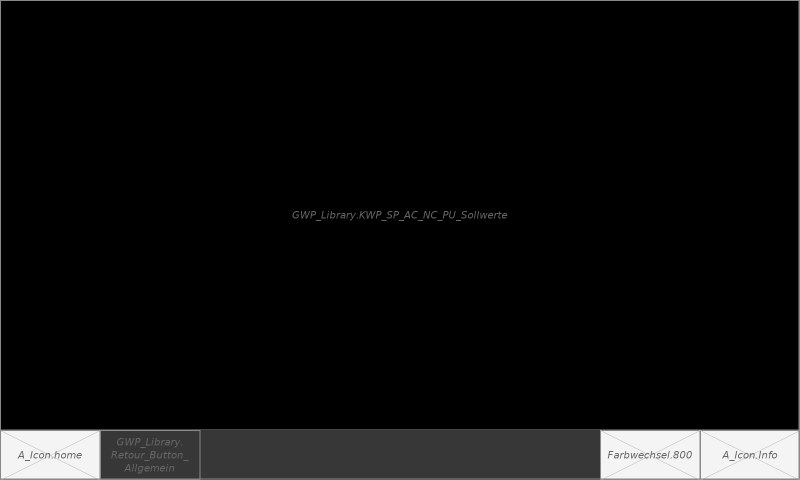
VISUALIZATION KWP_SP_AC_NC_PU_Sollwerte  // 800x480
    Frame (0,0 800x430)
        shows GWP_Library.KWP_SP_AC_NC_PU_Sollwerte(FB_KWP_SP_AC_NC := Main.KWP_SP_AC_NC_0)
    Frame (0,430 800x50)
        shows Fusszeile_50()
    Frame (100,430 100x50)
        shows GWP_Library.Retour_Button_Allgemein()
END_VISUALIZATION

// ---- VISUs/Betriebsarten/Wärmegewinnung/VD/VD_Sollwerte_zuruecksetzen.TcVIS
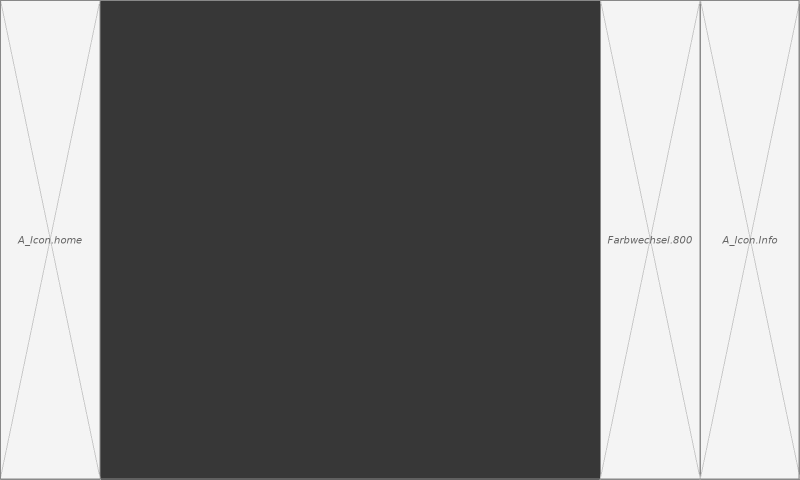
VISUALIZATION VD_Sollwerte_zuruecksetzen  // 800x480
    Frame (0,0 800x430)
        shows GWP_Library.VD_Sollwerte_zuruecksetzen(FB_VD := Main.VD_0)
    Frame (0,0 800x480)
        shows Fusszeile_50()
END_VISUALIZATION

// ---- VISUs/Betriebsarten/Wärmegewinnung/VD/VD.TcVIS
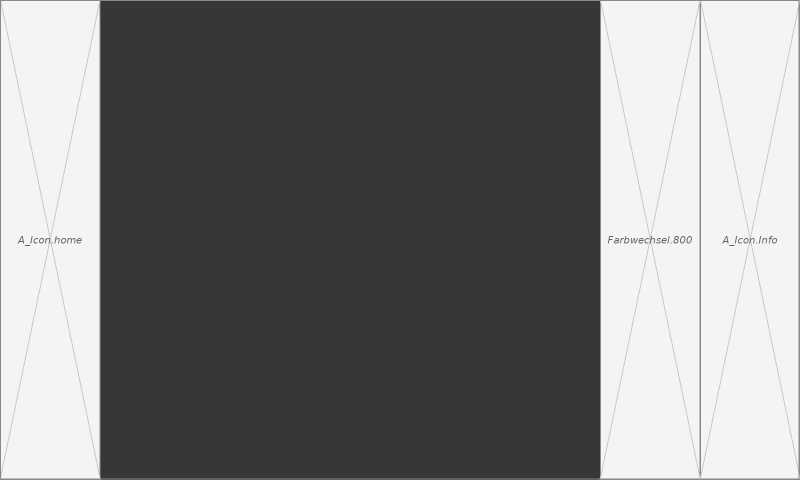
VISUALIZATION VD  // 800x480
    Frame (0,0 800x430)
        shows GWP_Library.VD(FB_VD := Main.VD_0)
    Frame (0,0 800x480)
        shows Fusszeile_50()
END_VISUALIZATION

// ---- VISUs/Betriebsarten/Wärmegewinnung/VD/VD_GW_Sollwerte.TcVIS
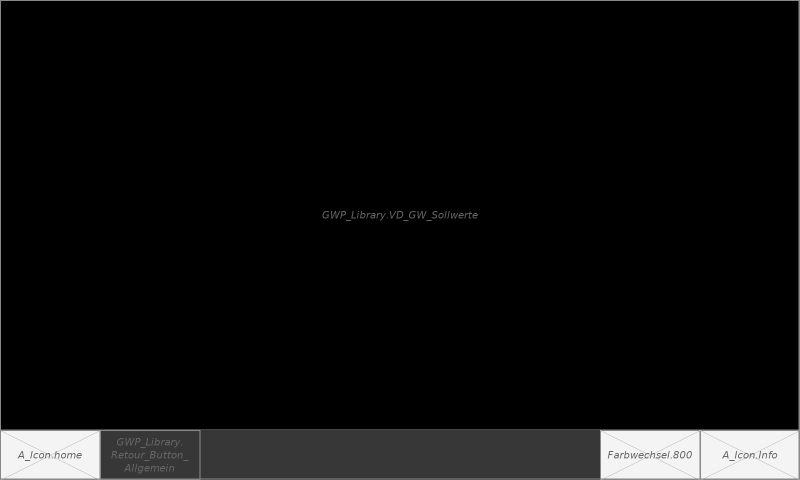
VISUALIZATION VD_GW_Sollwerte  // 800x480
    Frame (0,0 800x430)
        shows GWP_Library.VD_GW_Sollwerte(FB_VD := Main.VD_0)
    Frame (0,430 800x50)
        shows Fusszeile_50()
    Frame (100,430 100x50)
        shows GWP_Library.Retour_Button_Allgemein()
END_VISUALIZATION

// ---- VISUs/Betriebsarten/Wärmegewinnung/VD/VD_PU_Sollwerte.TcVIS
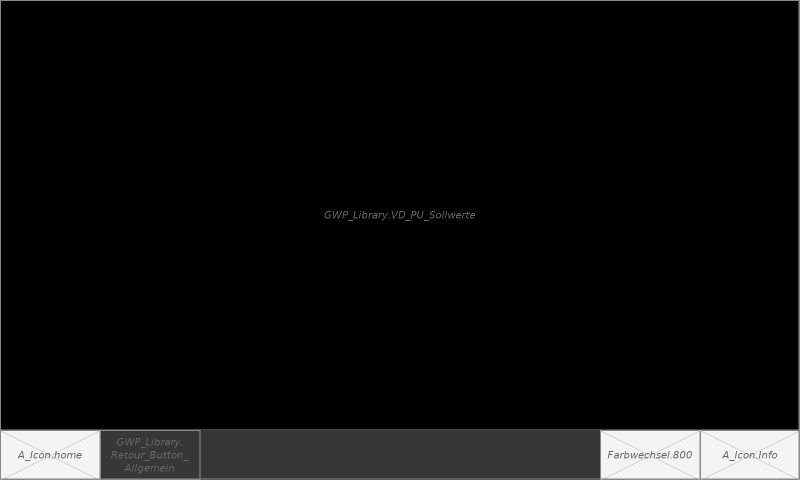
VISUALIZATION VD_PU_Sollwerte  // 800x480
    Frame (0,0 800x430)
        shows GWP_Library.VD_PU_Sollwerte(FB_VD := Main.VD_0)
    Frame (0,430 800x50)
        shows Fusszeile_50()
    Frame (100,430 100x50)
        shows GWP_Library.Retour_Button_Allgemein()
END_VISUALIZATION

// ---- VISUs/Betriebsarten/Wärmegewinnung/VD/VD_VTL_Sollwerte.TcVIS
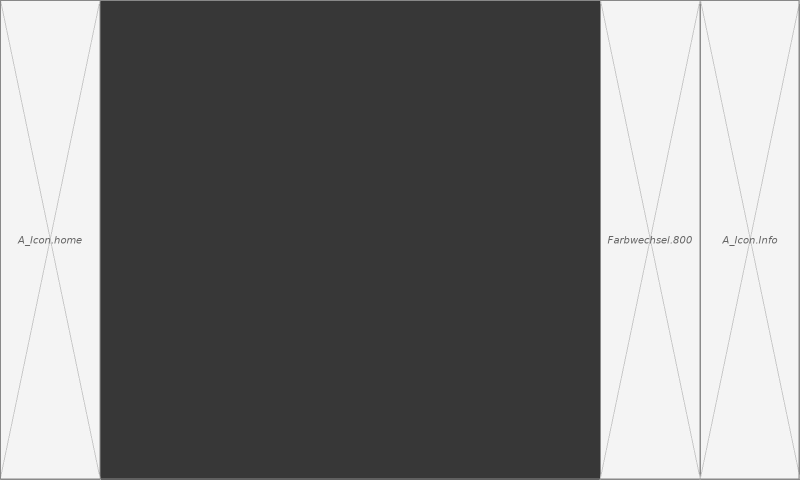
VISUALIZATION VD_VTL_Sollwerte  // 800x480
    Frame (0,0 800x430)
        shows GWP_Library.VD_VTL_Sollwerte(FB_VD := Main.VD_0)
    Frame (0,0 800x480)
        shows Fusszeile_50()
END_VISUALIZATION

// ---- VISUs/Betriebsarten/Wärmesenke/HWP_SP/HWP_SP.TcVIS
